Yaskawa INFORM job: FACE_S4.JBI

/JOB
//NAME FACE_S4
//POS
///NPOS 26,26,26,0,0,0
///TOOL 2
///POSTYPE PULSE
///PULSE
C00000=-121371,-17973,-37988,-31173,13272,35067
C00001=-121146,-12146,-50155,-33572,21711,37422
C00002=-120566,-9702,-52585,-34518,23996,37984
C00003=-120333,-8604,-53485,-34940,24912,38222
C00004=-120339,-4351,-50444,-34975,24986,38249
C00005=-120519,54946,2590,-33215,20736,36931
C00006=-120534,59103,6987,-32992,20094,36741
C00007=-120686,58394,7840,-32745,19352,36565
C00008=-121065,56831,10179,-32174,17465,36131
C00009=-121196,53724,22783,-30590,9788,34104
C00010=-122745,53813,23920,-27433,9078,34125
C00011=-122622,56537,10912,-28812,17063,35965
C00012=-122592,58038,8474,-29294,18937,36430
C00013=-120534,59103,6987,-32992,20094,36741
C00014=-122580,58724,7583,-29501,19674,36617
C00015=-123414,-10260,-51930,-30725,23420,37881
C00016=-123473,-12621,-49414,-29949,21189,37279
C00017=-123681,-18023,-36973,-27882,12480,35173
C00018=-120294,-18323,-35995,-22850,13259,33787
C00019=-120111,-13398,-48758,-24672,22325,35545
C00020=-120061,-11232,-51289,-25338,24592,36038
C00021=-120333,-8604,-53485,-34940,24912,38222
C00022=-120039,-10223,-52263,-25644,25533,36250
C00023=-120327,57401,9102,-24025,19740,35058
C00024=-120353,56036,11572,-23614,17820,34678
C00025=-120460,53740,25043,-22409,9420,33136
///TOOL 0
BC00000=77435
BC00001=77435
BC00002=77435
BC00003=77435
BC00004=77435
BC00005=77435
BC00006=77435
BC00007=77435
BC00008=77435
BC00009=77435
BC00010=86397
BC00011=86397
BC00012=86397
BC00013=77435
BC00014=86397
BC00015=86397
BC00016=86397
BC00017=86397
BC00018=86397
BC00019=86397
BC00020=86397
BC00021=77435
BC00022=86397
BC00023=86397
BC00024=86397
BC00025=86397
EC00000=-190707,176445
EC00001=-190707,176445
EC00002=-190707,176445
EC00003=-190707,176445
EC00004=-190707,176445
EC00005=-190707,176445
EC00006=-190707,176445
EC00007=-190707,176445
EC00008=-190707,176445
EC00009=-190707,176445
EC00010=-190707,176445
EC00011=-190707,176445
EC00012=-190707,176445
EC00013=-190707,176445
EC00014=-190707,176445
EC00015=-190707,176445
EC00016=-190707,176445
EC00017=-190707,176445
EC00018=-190707,176445
EC00019=-190707,176445
EC00020=-190707,176445
EC00021=-190707,176445
EC00022=-190707,176445
EC00023=-190707,176445
EC00024=-190707,176445
EC00025=-190707,176445
//INST
///DATE 2026/05/13 10:02
///ATTR SC,RW
///GROUP1 RB1,BS1
///GROUP2 ST1
NOP
'Face_s4
MEMOF
CLEAR MPF
'Path W7 (Root)
SSFTOF
MOVJ C00000 BC00000 VJ=100.00  +MOVJ EC00000 VJ=100.00
SMOVL C00001 BC00001 V=1000.0  +MOVJ EC00001
SMOVL C00002 BC00002 V=400.0  +MOVJ EC00002
SMOVL C00003 BC00003 T00001 V=10.0 PL=0  +MOVJ EC00003
SSFTOF
GETS PX001 $PX000
MEMON REC MPF#(1)
SMOVL C00004 BC00004 T00002 V=10.0  +MOVJ EC00004
SMOVL C00005 BC00005 T00003 V=10.0  +MOVJ EC00005
SMOVL C00006 BC00006 T00004 V=10.0  +MOVJ EC00006
MEMOF
GETS PX091 $PX000
SMOVL C00007 BC00007 V=400.0  +MOVJ EC00007
SMOVL C00008 BC00008 V=1000.0  +MOVJ EC00008
SMOVL C00009 BC00009 V=1000.0  +MOVJ EC00009
'EndPath W7 (Root)
'Path W9 (W7_Pass2)
SSFTOF
MOVJ C00010 BC00010 VJ=100.00  +MOVJ EC00010 VJ=100.00
SMOVL C00011 BC00011 V=1000.0  +MOVJ EC00011
SMOVL C00012 BC00012 V=400.0  +MOVJ EC00012
SREFP 1 C00013 BC00013  +REFP EC00013
SREFP 2 C00014 BC00014  +REFP EC00014
CALL JOB:LASKESFT-S1
SMOVL P091 V=23.0  +MOVJ EX091
MEMON BACKPLY MPF#(1)
SMOVL C00005 BC00005 T00003 V=10.0  +MOVJ EC00005
SMOVL C00004 BC00004 T00002 V=10.0  +MOVJ EC00004
SMOVL C00003 BC00003 T00001 V=10.0  +MOVJ EC00003
MEMOF
SMOVL C00015 BC00015 V=400.0  +MOVJ EC00015
SMOVL C00016 BC00016 V=1000.0  +MOVJ EC00016
SMOVL C00017 BC00017 V=100.0  +MOVJ EC00017
'EndPath W9 (W7_Pass2)
'Path W10 (W7_Pass3)
SSFTOF
MOVJ C00018 BC00018 VJ=100.00  +MOVJ EC00018 VJ=100.00
SMOVL C00019 BC00019 V=1000.0  +MOVJ EC00019
SMOVL C00020 BC00020 V=400.0  +MOVJ EC00020
SREFP 1 C00021 BC00021  +REFP EC00021
SREFP 2 C00022 BC00022  +REFP EC00022
CALL JOB:LASKESFT-S1
SMOVL P001 V=23.0  +MOVJ EX001
MEMON PLY MPF#(1)
SMOVL C00004 BC00004 T00002 V=10.0  +MOVJ EC00004
SMOVL C00005 BC00005 T00003 V=10.0  +MOVJ EC00005
SMOVL C00006 BC00006 T00004 V=10.0  +MOVJ EC00006
MEMOF
SMOVL C00023 BC00023 V=400.0  +MOVJ EC00023
SMOVL C00024 BC00024 V=1000.0  +MOVJ EC00024
SMOVL C00025 BC00025 V=1000.0  +MOVJ EC00025
'EndPath W10 (W7_Pass3)
END
